FUNCTION_BLOCK ABSTRACT Station IMPLEMENTS I_Station, I_Cyclic, I_Resettable, I_Object
VAR
	_IsClear : BOOL := TRUE;
	_Complete : BOOL;
	_Operating : BOOL;
	_Ready : BOOL := TRUE;
	_Position : LREAL := 0.0;
	_HasMover : BOOL;
	MoverArrive : R_TRIG;
	_MyMover : I_XtsMover;
END_VAR

{analysis -2}

METHOD PUBLIC  Cycle : HRESULT
VAR_INPUT
END_VAR
MoverArrive(CLK := _HasMover);
Operation();
IF MoverArrive.Q THEN
	_IsClear := FALSE;
	_Ready := FALSE;
	_Operating := TRUE;
	_Complete := FALSE;
END_IF

IF _Complete AND _HasMover AND_THEN _MyMover.AxisRef.NcToPlc.SetPos > _Position + 50  THEN
	_Ready := TRUE;
	_HasMover := FALSE;
	_IsClear := TRUE;
	_MyMover := 0;
END_IF
END_METHOD

//FB_Init is always available implicitly and it is used primarily for initialization.
//The return value is not evaluated. For a specific influence, you can also declare the
//methods explicitly and provide additional code there with the standard initialization
//code. You can evaluate the return value.
METHOD FB_Init: BOOL
VAR_INPUT
    bInitRetains: BOOL; // TRUE: the retain variables are initialized (reset warm / reset cold)
    bInCopyCode: BOOL;  // TRUE: the instance will be copied to the copy code afterward (online change)   
	Position : LREAL;
END_VAR
_Position := Position;
END_METHOD

METHOD HasMover : BOOL
VAR_INPUT
END_VAR
HasMover := _HasMover;
END_METHOD

METHOD IsClear : BOOL
IsClear := _IsClear;
END_METHOD

METHOD isComplete : BOOL
isComplete := _Complete;
END_METHOD

METHOD IsOperating : BOOL
IsOperating := _Operating;
END_METHOD

METHOD IsReady : BOOL
IsReady := _Ready;
END_METHOD

METHOD MyMover : HRESULT
VAR_INPUT
	mover : I_XtsMover;
END_VAR
IF mover = 0 THEN
	MyMover := -1;
	RETURN;
END_IF
IF _HasMover THEN
	MyMover := -2;
	RETURN;
END_IF
_HasMover := TRUE;
_MyMover := mover;
END_METHOD

METHOD PROTECTED ABSTRACT Operation : BOOL
VAR_INPUT
END_VAR
END_METHOD

PROPERTY Position : lreal
GET
Position := _Position;
END_GET
END_PROPERTY

METHOD RegisterWithParent
VAR_INPUT
	Parent	: I_HostObjects;
END_VAR
Parent.RegisterCyclic(THIS^);
END_METHOD

METHOD Reset : HRESULT
VAR_INPUT
END_VAR
_Complete := FALSE;
_IsClear := TRUE;
_Operating := FALSE;
_Ready := TRUE;
_HasMover := FALSE;
END_METHOD

END_FUNCTION_BLOCK

(* stored: Version 1.1.0.1
   POU Station: Id {506a1b5f-d283-4b99-9adf-318a9c36fdac}, SpecialFunc None
   Folder Status: Id {134213be-8709-40df-be5d-e58c074f6e63}
   Method Cycle: Id {718bc2ed-83e9-4df0-b688-ff0112cf7157}
   Method FB_Init: Id {65a20629-1237-49a2-826d-db1ec64ff183}
   Method HasMover: Id {1855cd52-e0ae-4354-8e0a-b89d5647c2a8}
   Method IsClear: Id {5a1d616a-dcb0-4a56-9caf-0526ba7a4fac}
   Method isComplete: Id {5a7054f2-4dbb-4c61-9bd3-b1648c0eccb5}
   Method IsOperating: Id {5d80dcb3-b05c-443a-91b8-3bed25c3df07}
   Method IsReady: Id {030f67f6-2ceb-4b14-bbf0-d64116218e04}
   Method MyMover: Id {cfa7f397-450b-4982-8373-384ee5df1767}
   Method Operation: Id {8b2af481-b3e4-47db-b897-3814deb87d2d}
   Property Position: Id {b89449d8-a019-4273-b99d-e422998e5fce}
   Get Get: Id {a533d869-853f-4701-aa82-723055982996}
   Method RegisterWithParent: Id {d8402b41-2440-40c0-90f4-c70380862930}
   Method Reset: Id {b49ff0e5-eb8b-49bd-befd-0bab45ac01fe} *)
